FUNCTION ST08X_TO_ARR08X (* this Function takes a a 8-BOOL Struct and makes a 8-BOOL Array *)
  (* Standard: 61499-1; Description: Copyright (c) 2024 HR Agrartechnik GmbH This program and the accompanying materials are made available under the terms of the Eclipse Public License 2.0 which is available at https://www.eclipse.org/legal/epl-2.0/ SPDX-License-Identifier: EPL-2.0 *)
  (* Version 1.0, 2024-02-22, Franz Höpfinger, HR Agrartechnik GmbH *)
  PACKAGE logiBUS::utils::conversion::str::converting;
  IMPORT eclipse4diac::core::TypeHash;
  IMPORT logiBUS::utils::conversion::types::ST08X;
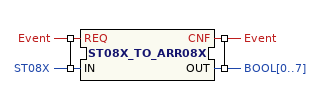
  EVENT_INPUT
    REQ WITH IN;
  END_EVENT
  EVENT_OUTPUT
    CNF WITH OUT;
  END_EVENT
  VAR_INPUT
    IN : logiBUS::utils::conversion::types::ST08X; (* ST08X Input *)
  END_VAR
  VAR_OUTPUT
    OUT : ARRAY [0..7] OF BOOL; (* ARR08X Output *)
  END_VAR
  BODY IN ST:
PACKAGE logiBUS::utils::conversion::str::converting;

IMPORT logiBUS::utils::conversion::types::ST08X;

(* this Function takes a a 8-BOOL Struct and makes a 8-BOOL Array *)
FUNCTION ST08X_TO_ARR08X

VAR_INPUT
	IN : ST08X; // ST08X Input
END_VAR

VAR_OUTPUT
	OUT : ARRAY[0..7] OF BOOL; // ARR08X Output
END_VAR

OUT[0] := IN.X_00;
OUT[1] := IN.X_01;
OUT[2] := IN.X_02;
OUT[3] := IN.X_03;
OUT[4] := IN.X_04;
OUT[5] := IN.X_05;
OUT[6] := IN.X_06;
OUT[7] := IN.X_07;

END_FUNCTION
  END_BODY
END_FUNCTION
